FUNCTION_BLOCK OUT_TEXT_S (* STRING Output to a TextArea-see OUT_TEXT *)
  (* Standard: 61499-1; Classification: GUI *)
  (* Version 0.1, 2002-05-03, JHC, Rockwell Automation, Made QI IV=true. *)
  (* Version 0.0, 2001-11-26, JHC, Rockwell Automation, Copied/modified from OUT_TEXT. *)
  (* Compiler header: package fb.rt.hmi; import java.awt.*; *)
  (* Compiler Java IBM VisualAge 3.0 *)
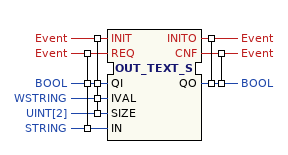
  EVENT_INPUT
    INIT WITH QI, IVAL, SIZE;
    REQ WITH QI, IN; (* Append IN to the TextArea *)
  END_EVENT
  EVENT_OUTPUT
    INITO WITH QO;
    CNF WITH QO;
  END_EVENT
  VAR_INPUT
    QI : BOOL := true;
    IVAL : WSTRING;
    SIZE : ARRAY [0..1] OF UINT := [10,20]; (* Rows,Columns *)
    IN : STRING;
  END_VAR
  VAR_OUTPUT
    QO : BOOL;
  END_VAR
END_FUNCTION_BLOCK
